// TIA Portal V20 export
TYPE "HMIAxisCtrl_typeGeneral"
TITLE = HMIAxisCtrl_typeGeneral
// Support: tech.team.motioncontrol@siemens.com 
// Fax: +49 (0) 9131/98-1297
   STRUCT
      axisType : DInt := 0;   // 1:SpeedAxis; 2:PosSyncAxis; 3:ExternalEncoder
      axisName : WString[24] := WSTRING#'No axis';   // Name of axis
      lengthUnit : UDInt;   // Unit for position
      velocityUnit : UDInt;   // Unit for velocity
      torqueForceUnit : UDInt;   // Unit for torque/Unit for force
      motionType : DInt := -1;   // Indication of axis or motion type: 0: Linear axis or motion 1: Rotary axis or motion
      encoderType : Int := 0;   // 1: Axis with incremental encoder; 2: Incremental external encoder; 3: Absolute external encoder or axis with absolute encoder
      moduloActive : Bool;   // TRUE: modulo active
      moduloLength : LReal;   // Modulo length
      limitBase : DInt := -1;   // Torque limiting. 0: Motor side; 1: Load side
      brakeExistent : Bool;   // TRUE: Brake existent
   END_STRUCT;
END_TYPE
